INTERFACE PUBLIC RunningStateCommands EXTENDS ClearedStateCommands

METHOD PUBLIC Stop
END_METHOD

END_INTERFACE

(* stored: Version 1.1.0.1, ProductVersion 3.1.4026.18
   Itf RunningStateCommands: Id {ac5a4eeb-897a-00c7-1851-dd2208974572}
   Method Stop: Id {3a91096d-df44-014e-055d-25aa25dac5d2} *)
